FUNCTION_BLOCK TExecution IMPLEMENTS IExecution 
VAR_INPUT
END_VAR
VAR_OUTPUT
END_VAR
VAR
	{attribute 'OPC.UA.DA' := '1'}
	State : TExecutionState := TExecutionState.Unknown;
	{attribute 'OPC.UA.DA' := '0'}
    _done : BOOL;       
	{attribute 'OPC.UA.DA' := '0'}
    _error : BOOL;      
	{attribute 'OPC.UA.DA' := '0'}
	_warning : BOOL;    
	{attribute 'OPC.UA.DA' := '0'}
    _aborted : BOOL;    
	{attribute 'OPC.UA.DA' := '0'}
    _errorId : UDINT;   
END_VAR

PROPERTY Aborted : BOOL
GET
Aborted := _aborted;
END_GET
SET
_aborted := Aborted;
END_SET
END_PROPERTY

PROPERTY Busy : BOOL
GET
Busy := State = TExecutionState.Busy;
END_GET
SET
END_SET
END_PROPERTY

PROPERTY Done : BOOL
GET
Done := _done;
END_GET
SET
_done := Done;
END_SET
END_PROPERTY

PROPERTY Error : BOOL
GET
Error := _error;
END_GET
SET
_error := Error;
END_SET
END_PROPERTY

PROPERTY ErrorId : UDINT
GET
ErrorId := _errorId;
END_GET
SET
_errorId := ErrorId;
END_SET
END_PROPERTY

PROPERTY Ready : BOOL;
GET
Ready := State = TExecutionState.Ready;
END_GET
SET
END_SET
END_PROPERTY

METHOD SetAborted
VAR_INPUT
END_VAR
_aborted := TRUE;
State := TExecutionState.Ready;
END_METHOD

METHOD SetBusy
VAR_INPUT
END_VAR
IF State = TExecutionState.Starting THEN
    State := TExecutionState.Busy;
END_IF
END_METHOD

METHOD SetDone 
VAR_INPUT
END_VAR
_done := TRUE;
State := TExecutionState.Ready;
END_METHOD

METHOD SetError
VAR_INPUT
	ErrorId : UDINT;
END_VAR
_error := TRUE;
_errorId := ErrorId;
State := TExecutionState.Error;
END_METHOD

METHOD SetReady
VAR_INPUT
END_VAR
// Clear results
_done := FALSE;
_error := FALSE;
_errorId := 0;
_aborted := FALSE;

State := TExecutionState.Ready;
END_METHOD

METHOD SetWarning
VAR_INPUT
END_VAR
_warning := TRUE;
State := TExecutionState.Ready;
END_METHOD

METHOD Start : BOOL
VAR_INPUT
END_VAR
IF State = TExecutionState.Ready OR 
    State = TExecutionState.Unknown THEN
    // Acq results
    _done := FALSE;
    _error := FALSE;
    _errorId := 0;
    _aborted := FALSE;
 
    State := TExecutionState.Starting;
 
    Start := TRUE;
END_IF
END_METHOD

PROPERTY Starting : BOOL
GET
Starting := State = TExecutionState.Starting ;
END_GET
SET
END_SET
END_PROPERTY

PROPERTY Status : TExecutionState
GET
Status := State;
END_GET
SET
State := Status;
END_SET
END_PROPERTY

PROPERTY Warning : BOOL
GET
Warning := _warning;
END_GET
SET
_warning := Warning;
END_SET
END_PROPERTY

END_FUNCTION_BLOCK

(* stored: Version 1.1.0.1, ProductVersion 3.1.4024.3
   POU TExecution: Id {c232843f-2ff3-4ae3-84e6-98da0146b076}, SpecialFunc None
   Property Aborted: Id {63541121-7ea3-43b2-9ae4-cbf326229b7c}
   Get Get: Id {95435308-f8a9-4b0f-95a7-ec8ac4d06f37}
   Set Set: Id {8b9942ad-18e0-4465-98ac-3ccad9137aed}
   Property Busy: Id {a3f02e88-03be-4951-a37c-c9d808c3ee62}
   Get Get: Id {bceb8f9b-b9ee-4a8e-882e-76cd043ea681}
   Set Set: Id {c6c03b95-8b42-4736-9ce3-9836c5ca9915}
   Property Done: Id {09d28897-2204-4f66-a4a3-b9063439c371}
   Get Get: Id {97769fc5-971f-4cbe-81a7-7467e40db7c8}
   Set Set: Id {76d0680b-e3ed-429b-9cd5-e9cda76fb027}
   Property Error: Id {02de8373-4279-4f3a-8fac-086f215450b4}
   Get Get: Id {807c373f-05a3-4ad7-a428-9387dbad42b7}
   Set Set: Id {f6e59a86-6b55-4a7f-9a73-69d38964f84c}
   Property ErrorId: Id {26a5bb13-b25d-440e-95e8-2ce3ff8fb464}
   Get Get: Id {17ec13f1-8b01-4021-bfc0-bb1a1a91d1f2}
   Set Set: Id {c2e2bed9-b8ff-47b4-a142-ef4431d6fbec}
   Property Ready: Id {bf2a027e-dcb8-4505-a0e4-2adde474bd26}
   Get Get: Id {070109f7-939a-43ba-aeba-d4844ab81208}
   Set Set: Id {471c697d-888e-4b80-8690-c5c818286aa4}
   Method SetAborted: Id {10747d03-e24d-41e7-9827-e00e9d1be62c}
   Method SetBusy: Id {1dae19c1-6c16-43c0-b1a9-04eaeae3319e}
   Method SetDone: Id {63e34279-45bb-4d75-ae9f-096e5adac110}
   Method SetError: Id {21085a73-cb46-40d6-92f7-fea024288e0b}
   Method SetReady: Id {77cd0482-f8ed-431c-8a95-4405ea835cf0}
   Method SetWarning: Id {ac5d607e-0cc8-40c7-93f3-c283687c2812}
   Method Start: Id {f2e1fefe-a947-4e6e-b485-10f29c05c92b}
   Property Starting: Id {28851dbe-824c-4e36-807b-5f37db759fa2}
   Get Get: Id {89b3cac5-cec5-498e-bebe-43c703b8a74d}
   Set Set: Id {aaa40f74-2661-4c48-8595-6bca47f72bd8}
   Property Status: Id {82a80d98-c72b-4a22-ae32-f52f84505555}
   Get Get: Id {df009eef-510b-492f-a59f-414253a85df9}
   Set Set: Id {16782c7c-5389-45d1-a065-c864880c5fc6}
   Property Warning: Id {ccc41633-9723-4790-bed6-ffa5e79fc332}
   Get Get: Id {e811a603-305b-43a0-a4fb-0e29e56d27e8}
   Set Set: Id {0766741c-8ba5-4139-a5c0-a04c08cbf85a} *)
